Fanuc KAREL source: NC0089.KL

-- PROVISIONAL review KL for V1013-1; original PC SHA256 69c15732cdf82d19a94a46e70be86278424f829d88b554ce3f1eb6ac4b3022e3
-- Incomplete behavior may be omitted. Consult companion uncertainty JSON. Do not deploy.
PROGRAM NC0089
%NOLOCKGROUP
-- UNRESOLVED_LOCAL_POOL 5 cells at code offset 3; source declarations unknown
-- DIRECT_LOCAL_WORD_ACCESS alone does not prove INTEGER, REAL, or BOOLEAN
BEGIN
  -- UNRESOLVED_PC offsets 0-8; opcodes 2B,2C,7B
  -- UNRESOLVED_PC offsets 13-20; opcodes 9D,23
  -- UNRESOLVED_PC offsets 25-38; opcodes 21,9D,57,79
  -- UNRESOLVED_PC offsets 43-60; opcodes 21,40,41,42
  -- UNRESOLVED_PC offsets 65-94; opcodes 9D,23,9E,2E,22,7A
  -- UNRESOLVED_PC offsets 99-116; opcodes 21,2E,59,79
  -- UNRESOLVED_PC offsets 121-134; opcodes 21,9D,57,79
  -- UNRESOLVED_PC offsets 139-156; opcodes 21,40,41,42
  -- UNRESOLVED_PC offsets 161-190; opcodes 9D,23,9E,2E,22,7A
  -- UNRESOLVED_PC offsets 195-212; opcodes 21,2E,59,79
  -- UNRESOLVED_PC offsets 217-230; opcodes 21,9D,57,79
  -- UNRESOLVED_PC offsets 235-252; opcodes 21,40,41,42
  -- UNRESOLVED_PC offsets 257-286; opcodes 9D,23,9E,2E,22,7A
  -- UNRESOLVED_PC offsets 291-308; opcodes 21,2E,59,79
  -- UNRESOLVED_PC offsets 313-326; opcodes 21,9D,57,79
  -- UNRESOLVED_PC offsets 331-348; opcodes 21,40,41,42
  -- UNRESOLVED_PC offsets 353-382; opcodes 9D,23,9E,2E,22,7A
  -- UNRESOLVED_PC offsets 387-401; opcodes 21,9D,52,23
  -- UNRESOLVED_PC offsets 406-437; opcodes 20,2C,23,7A,40,41,42
  -- UNRESOLVED_PC offsets 442-466; opcodes 21,2E,52,23,7A,43
  -- UNRESOLVED_PC offsets 471-489; opcodes 21,2E,52,23
  -- UNRESOLVED_PC offsets 499-504; opcodes 7A
  -- UNRESOLVED_PC offsets 509-527; opcodes 21,2E,52,23
  -- UNRESOLVED_PC offsets 537-542; opcodes 7A
  -- UNRESOLVED_PC offsets 547-578; opcodes 20,2C,23,7A,40,41,42
  -- UNRESOLVED_PC offsets 583-607; opcodes 21,2E,52,23,7A,43
  -- UNRESOLVED_PC offsets 612-630; opcodes 21,2E,52,23
  -- UNRESOLVED_PC offsets 640-645; opcodes 7A
  -- UNRESOLVED_PC offsets 650-668; opcodes 21,2E,52,23
  -- UNRESOLVED_PC offsets 678-683; opcodes 7A
  -- UNRESOLVED_PC offsets 688-719; opcodes 20,2C,23,7A,40,41,42
  -- UNRESOLVED_PC offsets 724-748; opcodes 21,2E,52,23,7A,43
  -- UNRESOLVED_PC offsets 753-771; opcodes 21,2E,52,23
  -- UNRESOLVED_PC offsets 781-786; opcodes 7A
  -- UNRESOLVED_PC offsets 791-809; opcodes 21,2E,52,23
  -- UNRESOLVED_PC offsets 819-824; opcodes 7A
  -- UNRESOLVED_PC offsets 829-860; opcodes 20,2C,23,7A,40,41,42
  -- UNRESOLVED_PC offsets 865-889; opcodes 21,2E,52,23,7A,43
  -- UNRESOLVED_PC offsets 894-912; opcodes 21,2E,52,23
  -- UNRESOLVED_PC offsets 922-927; opcodes 7A
  -- UNRESOLVED_PC offsets 932-950; opcodes 21,2E,52,23
  -- UNRESOLVED_PC offsets 960-964; opcodes 7F
  -- UNRESOLVED_PC offsets 969-973; opcodes 27,AA
  -- UNRESOLVED_PC offsets 978-982; opcodes 7F
END NC0089
